RoboDK station: picknplace.rdk

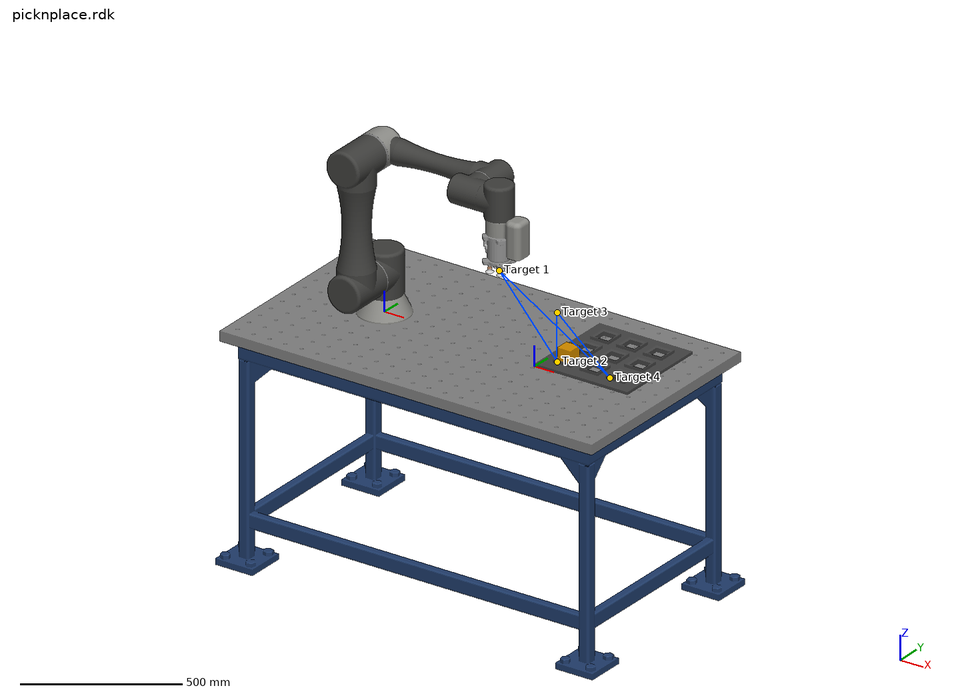
[picture v0: the station drawn from its stored meshes, robots at their saved joint values, targets as dots, program paths as lines]
Station picknplace (saved by RoboDK 5.9.2). Poses are relative to the parent item; angles as X-Y-Z fixed-axis rotations.
  - frame TM5-900 Base at (0, 0, 0) mm
    - robot TM5-900: 6 axes, payload 4 kg, reach 900 mm, repeatability 0.1 mm, weight 30 kg
        modified DH rows (alpha deg, a mm, theta deg, d mm): 0, 0, 0, 145.2; 90, 0, 90, 0; 0, 429, 0, 0; 0, 411, -90, 122.3; -90, 0, 0, 106.5; 90, 0, 180, 114.15
        joint limits [-360, -180, -155, -180, -180, -270] to [360, 180, 155, 180, 180, 270]; home [0, 0, 90, -90, 90, 0]; saved at [0, 0, 90, 0, 90, 0]
      - tool SMC ZXP7A01-ZP25C-X1 Vacuum Gripper, TCP at (0, 0, 125) mm, size 88 x 106.8 x 127.9 mm
  - object Table 1400x800x800mm at (0, 0, 0) mm, size 1420 x 820 x 800 mm, geometry from Table-1400x800x800mm.sld
  - frame Frame 2 at (600, -50, 0) mm
    - target Target 1 (Cartesian target) at (-82.5, -72.3, 335.05) mm, rotated rx 180 ry 0 rz 90 deg; joints [0, 0, 90, 0, 90, 0] of TM5-900
    - target Target 2 (Cartesian target) at (50, 50, 10) mm, rotated rx 180 ry 0 rz 90 deg; joints [10.845, 30.56, 99.672, -40.232, 90, 10.845] of TM5-900
    - target Target 3 (Cartesian target) at (50, 50, 180) mm, rotated rx 180 ry 0 rz 90 deg; joints [10.845, 19.365, 89.189, -18.554, 90, 10.845] of TM5-900
    - target Target 4 (Cartesian target) at (250, 50, 10) mm, rotated rx 180 ry 0 rz 90 deg; joints [8.273, 54.634, 55.928, -20.562, 90, 8.273] of TM5-900
    - object Pallete  at (0, 0, 0) mm, size 350 x 350 x 20 mm, geometry from Pallete .step
    - object Cube 50mm at (50, 50, 10) mm, size 50 x 50 x 50 mm, geometry from Cube-50mm.sld
  - program Prog1 (9 instructions, listed below)
  - program Prog2 (1 instructions, listed below)
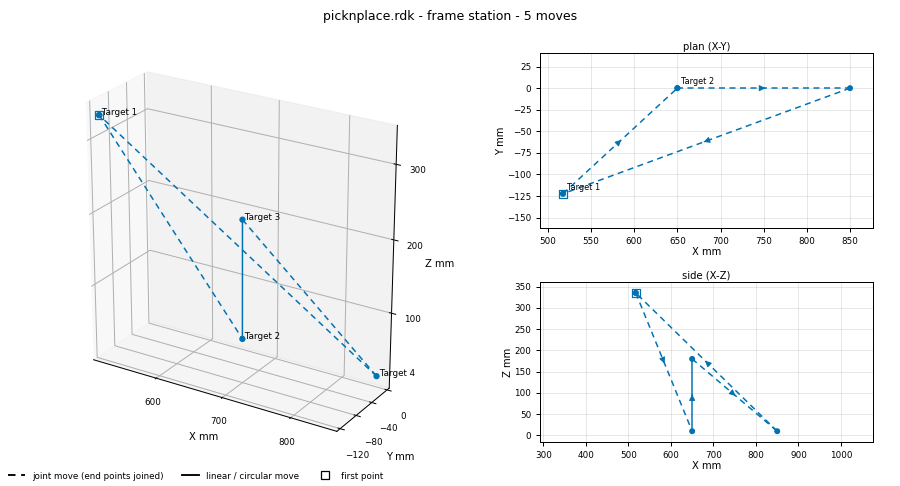
[picture p0: tool path of picknplace.rdk in frame station, 5 of 5 moves have a stored position in this frame; points joined in program order, loops and branches not executed]

--- program Prog1 (robot TM5-900) ---
  Set Ref.: Frame 2
  Set Tool: SMC ZXP7A01-ZP25C-X1 Vacuum Gripper
  MoveJ (Target 1)
  MoveJ (Target 2)
  Attach to SMC ZXP7A01-ZP25C-X1 Vacuum Gripper
  MoveL (Target 3)
  MoveJ (Target 4)
  Detach from SMC ZXP7A01-ZP25C-X1 Vacuum Gripper
  MoveJ (Target 1)

--- program Prog2 (robot TM5-900) ---
  Replace objects
